Staubli VAL3: countBool.pgx

public program countBool(bool& x_bInput[], num& x_nResult)
  local num l_nLength
  local num l_nElement
begin

  l_nLength = size(x_bInput)
  x_nResult = 0

  for l_nElement = 0 to l_nLength-1
    if x_bInput[l_nElement] == true
      x_nResult = x_nResult+1
    endIf
  endFor

end
